FUNCTION_BLOCK FB_FirePyroModeCommand IMPLEMENTS I_Command
VAR
	refFlameCannon : REFERENCE TO FB_FlameCannon;
END_VAR

METHOD Execute
IF (__ISVALIDREF(THIS^.refFlameCannon)) THEN
	THIS^.refFlameCannon.On();
	THIS^.refFlameCannon.SetLevel(95.00);
END_IF
END_METHOD

METHOD FB_init : BOOL
VAR_INPUT
	bInitRetains 	: BOOL; // if TRUE, the retain variables are initialized (warm start / cold start)
	bInCopyCode 	: BOOL;  // if TRUE, the instance afterwards gets moved into the copy code (online change)
	refFlameCannon 	: REFERENCE TO FB_FlameCannon;
END_VAR
IF (__ISVALIDREF(refFlameCannon)) THEN
	THIS^.refFlameCannon REF= refFlameCannon;
ELSE
	THIS^.refFlameCannon REF= 0;
END_IF
END_METHOD

END_FUNCTION_BLOCK

(* stored: Version 1.1.0.1, ProductVersion 3.1.4022.18
   POU FB_FirePyroModeCommand: Id {b25aa89e-c419-4dc6-816c-0a0cfa2a379f}, SpecialFunc None
   Method Execute: Id {7eca64eb-b034-4d04-a9ed-f8ce686e7d45}
   Method FB_init: Id {6af10b78-705f-4e22-a7a6-661f4685e583} *)
